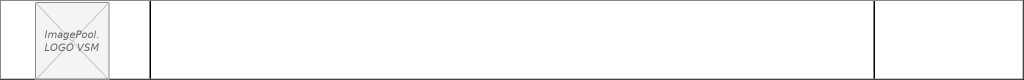
VISUALIZATION Header  // 1024x80
    Rectangle (0,0 150x80)
    Rectangle (150,0 724x80)
    Rectangle (874,0 150x80)
    Image (35,2 74x78), image: ImagePool.LOGO VSM
END_VISUALIZATION

(* stored: Version 1.1.0.1, ProductVersion 3.1.4024.12
   Visu Header: Id {5b9f1c8e-c458-4c21-a8f2-47c0224fae2b} *)
